FUNCTION_BLOCK AUI_DEMUX_4 (* Event demultiplexer with AUI adapter input instead of plain EI+K (generic FB) *)
  (* Standard: 61499-1 Annex A; Description: Copyright (c) 2017 fortiss GmbH This program and the accompanying materials are made available under the terms of the Eclipse Public License 2.0 which is available at https://www.eclipse.org/legal/epl-2.0/ SPDX-License-Identifier: EPL-2.0 *)
  (* Version 1.0, 2026-09-10, Franz Höpfinger, HR Agrartechnik GmbH, AUI adapter variant of E_DEMUX_4 *)
  PACKAGE adapter::events::unidirectional;
  {SET_ATTRIBUTE(eclipse4diac::core::GenericClassName, 'GEN_AUI_DEMUX')}
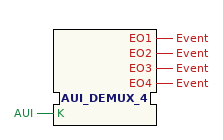
  EVENT_OUTPUT
    EO1; (* Output, demultiplexed from EI when K=0 *)
    EO2; (* Output, demultiplexed from EI when K=1 *)
    EO3; (* Output, demultiplexed from EI when K=2 *)
    EO4; (* Output, demultiplexed from EI when K=3 *)
  END_EVENT
  SOCKETS
    K : adapter::types::unidirectional::AUI; (* Event index *)
  END_SOCKETS
END_FUNCTION_BLOCK
